FUNCTION_BLOCK FB_HE_SATT_FilterCombinationToTransmission_Test EXTENDS FB_TestSuite


GivenCombinationExpectCorrectTransmission();


METHOD PRIVATE GivenCombinationExpectCorrectTransmission
VAR
    
END_VAR

TEST('GivenCombinationExpectCorrectTransmission');



TEST_FINISHED();
END_METHOD

END_FUNCTION_BLOCK

(* stored: Version 1.1.0.1
   POU FB_HE_SATT_FilterCombinationToTransmission_Test: Id {56e703d8-4a85-4aec-be27-be94d09287a6}, SpecialFunc None
   Method GivenCombinationExpectCorrectTransmission: Id {33419f85-4452-4060-ae9f-55feccaf063b} *)
